# B&R Automation Studio project lab1
Automation Studio 4.5.2.102

## Configuration Config1

### Hardware
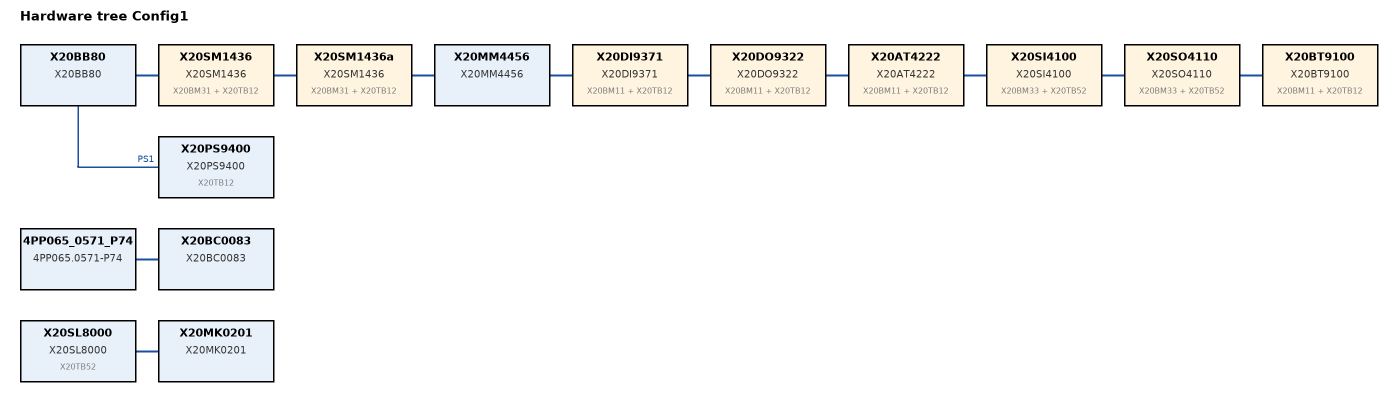
```
4PP065_0571_P74 : 4PP065.0571-P74 v1.1.2.0
  Connector IF5:
    ActivateDevice = 1
    Mode = Manual
    InternetAddress = 10.0.1.10
    SubnetMask = 255.255.255.0
  ConfigurationID = labBR
  Simulation = 1
X20AT4222 : X20AT4222 v1.2.3.0  [SS1 -> X20TB12e.SS; SL -> X20BM11b.SL1]
X20BB80 : X20BB80 v1.0.2.0
X20BC0083 : X20BC0083 v2.7.0.0  [PLK1 -> 4PP065_0571_P74.IF4 [Cable Type=PowerlinkCable, Length=10, Version=1.0.0.2]; SL -> X20BB80.SL1]
X20BM11 : X20BM11 v1.0.0.1  [X2X1 -> X20MM4456.X2X2]
X20BM11a : X20BM11 v1.0.0.1  [X2X1 -> X20BM11.X2X2]
X20BM11b : X20BM11 v1.0.0.1  [X2X1 -> X20BM11a.X2X2]
X20BM11c : X20BM11 v1.0.0.1  [X2X1 -> X20BM33a.X2X2]
X20BM31 : X20BM31 v1.0.0.1  [X2X1 -> X20BB80.IF1]
X20BM31a : X20BM31 v1.0.0.1  [X2X1 -> X20BM31.X2X2]
X20BM33 : X20BM33 v1.0.0.4  [X2X1 -> X20BM11b.X2X2]
X20BM33a : X20BM33 v1.0.0.4  [X2X1 -> X20BM33.X2X2]
X20BT9100 : X20BT9100 v1.0.3.0  [SS1 -> X20TB12f.SS; SL -> X20BM11c.SL1]
X20DI9371 : X20DI9371 v1.0.2.0  [SS1 -> X20TB12c.SS; SL -> X20BM11.SL1]
X20DO9322 : X20DO9322 v1.0.3.0  [SS1 -> X20TB12d.SS; SL -> X20BM11a.SL1]
X20MK0201 : X20MK0201 v1.0.0.0  [SL -> X20SL8000.SL1]
X20MM4456 : X20MM4456 v1.1.5.0  [X2X1 -> X20BM31a.X2X2]
X20PS9400 : X20PS9400 v1.0.2.4  [SS1 -> X20TB12.SS; PS -> X20BB80.PS1]
X20SI4100 : X20SI4100 v1.10.1.1  [SS1 -> X20TB52a.SS; SL -> X20BM33.SL1]
X20SL8000 : X20SL8000 v1.6.5.1  [SS1 -> X20TB52.SS]
X20SM1436 : X20SM1436 v1.4.2.1  [SS1 -> X20TB12a.SS; SL -> X20BM31.SL1]
  FunctionModel = Standard
X20SM1436a : X20SM1436 v1.4.2.1  [SS1 -> X20TB12b.SS; SL -> X20BM31a.SL1]
  FunctionModel = Standard
X20SO4110 : X20SO4110 v1.10.1.1  [SS1 -> X20TB52b.SS; SL -> X20BM33a.SL1]
  SafeModuleID = 3
X20TB12 : X20TB12 v1.0.0.0
X20TB12a : X20TB12 v1.0.0.0
X20TB12b : X20TB12 v1.0.0.0
X20TB12c : X20TB12 v1.0.0.0
X20TB12d : X20TB12 v1.0.0.0
X20TB12e : X20TB12 v1.0.0.0
X20TB12f : X20TB12 v1.0.0.0
X20TB52 : X20TB52 v1.0.0.1
X20TB52a : X20TB52 v1.0.0.1
X20TB52b : X20TB52 v1.0.0.1
```

## Logical view

### Global.var - Global variables
```iecst
VAR
	count : USINT;
END_VAR
```

### Package Logical/Libraries - Global libraries

### Library Logical/Libraries/MotorCtrl (ANSIC)

#### MotorCtrl.fun - Exported functions and function blocks
```iecst
FUNCTION_BLOCK FB_Integrator
	VAR_INPUT
		in : REAL;
	END_VAR
	VAR_OUTPUT
		out : REAL;
	END_VAR
	VAR
		dt : REAL;
	END_VAR
END_FUNCTION_BLOCK

FUNCTION_BLOCK FB_Motor
	VAR_INPUT
		u : REAL;
	END_VAR
	VAR_OUTPUT
		w : REAL;
		phi : REAL;
	END_VAR
	VAR
		integrator : FB_Integrator;
		Tm : REAL;
		ke : REAL;
		dt : REAL;
	END_VAR
END_FUNCTION_BLOCK

FUNCTION_BLOCK FB_Regulator
	VAR_INPUT
		e : REAL;
		e_prev : REAL;
	END_VAR
	VAR_OUTPUT
		u : REAL;
	END_VAR
	VAR
		u_raw : REAL;
		count : USINT;
		k_p : REAL;
		k_i : REAL;
		integrator : FB_Integrator;
		iyOld : REAL;
		max_abs_value : REAL;
		dt : REAL;
	END_VAR
END_FUNCTION_BLOCK
```

#### FB_Regulator.c
```c
#include <bur/plctypes.h>
#ifdef __cplusplus
	extern "C"
	{
#endif
#include "MotorCtrl.h"
#ifdef __cplusplus
	};
#endif
/* TODO: Add your comment here */
void FB_Regulator(struct FB_Regulator* inst)
{
	// Интегратор в прямой цепи
	/*inst->u += (inst->k_p * inst->e <= inst->max_abs_value ? inst->k_p * inst->e : inst->max_abs_value) +
		inst->k_i * inst->dt * inst->e_prev -
		(inst->k_p * inst->e_prev <= inst->max_abs_value ? inst->k_p * inst->e_prev : inst->max_abs_value);

	//Ограничение напряжения
	if (inst->u > inst->max_abs_value)
		inst->u = inst->max_abs_value;
	*/

	// Интегратор в обратной цепи
	inst->u_raw = (inst->k_p * inst->e <= inst->max_abs_value ? inst->k_p * inst->e : inst->max_abs_value) -
		(inst->k_p * inst->e_prev <= inst->max_abs_value ? inst->k_p * inst->e_prev : inst->max_abs_value) +
		inst->k_i * inst->dt * inst->e + (inst->u - inst->iyOld);

	if (inst->u_raw <= inst->max_abs_value)
		inst->u = inst->u_raw;
	else
	{
		inst->u_raw = (inst->u_raw + inst->max_abs_value) / 2;  //truncating-scheme input
		inst->u = inst->max_abs_value;
	}
	inst->iyOld = inst->u - inst->u_raw;  //updating old truncating-scheme output
}
```

#### FB_Motor.c
```c
#include <bur/plctypes.h>
#ifdef __cplusplus
	extern "C"
	{
#endif
#include "MotorCtrl.h"
#ifdef __cplusplus
	};
#endif
/* TODO: Add your comment here */
void FB_Motor(struct FB_Motor* inst)
{
	//direct circuit
	/*inst->w = inst->w * (inst->Tm - inst->dt) / inst->Tm +
		inst->u * inst->dt / (inst->ke * inst->Tm);*/

	//feedback circuit
	inst->w = inst->w * inst->Tm / (inst->Tm + inst->dt) +
		inst->u * inst->dt / (inst->ke * (inst->Tm + inst->dt));

//	inst->integrator.in = (inst->u / inst->ke - inst->w) / inst->Tm;
//	FB_Integrator(&inst->integrator);
//	inst->w = inst->integrator.out;

//	inst->integrator.in = inst->w;
//	FB_Integrator(&inst->integrator);
//	inst->phi = inst->integrator.out;

}
```

#### FB_Integrator.c
```c
#include <bur/plctypes.h>
#ifdef __cplusplus
	extern "C"
	{
#endif
#include "MotorCtrl.h"
#ifdef __cplusplus
	};
#endif
/* TODO: Add your comment here */
void FB_Integrator(struct FB_Integrator* inst)
{
	inst->out += inst->in * inst->dt;
}
```

### Program Logical/Prog1 (ANSIC)

#### Variables.var
```iecst
VAR
	fb_regulator : FB_Regulator; (*Рассогласование между задающим воздействием и реальной скоростью рассогласование между задающим воздействием и реальной скоростью рассогласование между задающим воздействием и реальной скоростью вращения вала ДПТ [об/мин]*)
	fb_motor : FB_Motor; (*Напряжение, подаваемое на вход ДПТ [В]	*)
	speed : REAL; (*Уставка по скорости*)
	enable : BOOL; (*Включение системы управления*)
	mot_prev : REAL; (*Предыдущее значение для двигателя*)
	reg_prev : REAL; (*Предыдущее значение для регулятора*)
	fb_motor2 : FB_Motor;
END_VAR
```

#### Main.c
```c
#include <bur/plctypes.h>

#ifdef _DEFAULT_INCLUDES
	#include <AsDefault.h>
#endif

void _INIT ProgramInit(void)
{
	enable = 0;

	speed = count = 0;

	fb_motor.dt = fb_regulator.dt = 0.002;
	fb_motor2.dt = 0.002;

	fb_regulator.k_p = 0.0064;
	fb_regulator.k_i = 0.16;
	fb_regulator.max_abs_value = 24;

	fb_motor.Tm = fb_regulator.k_p / fb_regulator.k_i;
	fb_motor.ke = 3 * fb_motor.dt * fb_regulator.k_i;

	fb_motor2.Tm = fb_regulator.k_p / fb_regulator.k_i;
	fb_motor2.ke = 3 * fb_motor2.dt * fb_regulator.k_i;
}

void _CYCLIC ProgramCyclic(void)
{
	if (count > 1)
	enable = 1;

	if (enable)
	{
		//step function (10 secs period)
		if (count % 50 == 0){
			speed = speed == 0 ? 2000 : 0;
		}
		//processing system's output (integrator link in direct circuit)
		/*fb_regulator.e = speed - fb_motor.w;
		fb_regulator.e_prev = reg_prev;
		FB_Regulator(&fb_regulator);
		fb_motor.u = mot_prev;
		FB_Motor(&fb_motor);*/

		//processing system's output (integrator link in feedback circuit)
		fb_regulator.e = speed - fb_motor.w;
		fb_regulator.e_prev = reg_prev;
		fb_regulator.count = count;
		FB_Regulator(&fb_regulator);
		fb_motor.u = fb_regulator.u;
		//fb_motor.u = fb_motor.ke*speed;
		FB_Motor(&fb_motor);

		// Для второго двигателя
		fb_motor2.u = fb_motor2.ke*speed;
		FB_Motor(&fb_motor2);

		//(current input on step [k] equals previous input on step [k + 1])
		reg_prev = fb_regulator.e;
		mot_prev = fb_regulator.u;
	}

	//updating state
	count++;
}

void _EXIT ProgramExit(void)
{

}
```

Listed in the project but not available here: Logical/Global.typ, Logical/Libraries/MotorCtrl/Types.typ, Logical/Libraries/MotorCtrl/Constants.var
